FUNCTION_BLOCK logiBUS_PI_ID (* Input service interface function block for double word input data *)
  (* Description: Copyright (c) 2017 fortiss GmbH, HR Agrartechnik GmbH This program and the accompanying materials are made available under the terms of the Eclipse Public License 2.0 which is available at https://www.eclipse.org/legal/epl-2.0/ SPDX-License-Identifier: EPL-2.0 if ImpulseDelta = 0, then TimeDelta cannot be 0. set TimeDelta to 16#FFFFFFFF to deactivate cyclic processing, and onyl indicate Changes in Value. *)
  (* Version 1.0, 2017-03-20, Monika Wenger, fortiss GmbH, initial API and implementation and/or initial documentation *)
  PACKAGE logiBUS::io::PI;
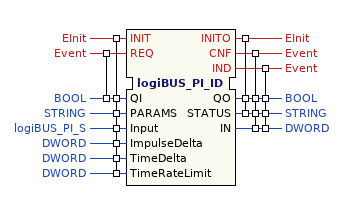
  EVENT_INPUT
    INIT : EInit WITH QI, PARAMS, Input, ImpulseDelta, TimeDelta, TimeRateLimit; (* Service Initialization *)
    REQ WITH QI; (* Service Request *)
  END_EVENT
  EVENT_OUTPUT
    INITO : EInit WITH QO, STATUS; (* Initialization Confirm *)
    CNF WITH QO, STATUS, IN; (* Confirmation of Requested Service *)
    IND WITH QO, STATUS, IN; (* Indication from Resource *)
  END_EVENT
  VAR_INPUT
    QI : BOOL; (* Event Input Qualifier *)
    PARAMS : STRING; (* Service Parameters *)
    Input : logiBUS::io::PI::logiBUS_PI_S := logiBUS_PI::Invalid; (* Identify the Input Input_I1..I8 *)
    ImpulseDelta : DWORD; (* After How many Impulses an IND *)
    TimeDelta : DWORD := 250; (* After How many ms an IND *)
    TimeRateLimit : DWORD := 100; (* Maximum 1 IND in how many ms. (< delta) *)
  END_VAR
  VAR_OUTPUT
    QO : BOOL; (* Event Output Qualifier *)
    STATUS : STRING; (* Service Status *)
    IN : DWORD; (* Input data from resource *)
  END_VAR
END_FUNCTION_BLOCK
